FUNCTION_BLOCK CylinderVSensValve (* Composite Function Block Type *)
  (* Standard: 61499-2 *)
  (* Version 0.0, 5/29/2016, Andrei, nxtControl GmbH, template *)
  PACKAGE Main;
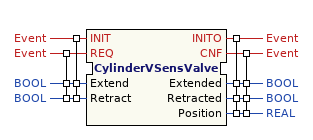
  EVENT_INPUT
    INIT WITH Extend, Retract; (* Initialization Request *)
    REQ WITH Extend, Retract; (* Normal Execution Request *)
  END_EVENT
  EVENT_OUTPUT
    INITO WITH Extended, Retracted, Position; (* Initialization Confirm *)
    CNF WITH Extended, Retracted, Position; (* Execution Confirmation *)
  END_EVENT
  VAR_INPUT
    Extend : BOOL; (* Input event qualifier *)
    Retract : BOOL;
  END_VAR
  VAR_OUTPUT
    Extended : BOOL; (* Output event qualifier *)
    Retracted : BOOL;
    Position : REAL;
  END_VAR
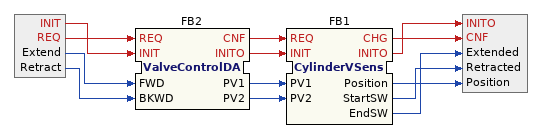
  FBS
    FB2 : ValveControlDA;
    FB1 : CylinderVSens;
  END_FBS
  EVENT_CONNECTIONS
    REQ TO FB2.REQ;
    INIT TO FB2.INIT;
    FB2.CNF TO FB1.REQ;
    FB1.CHG TO CNF;
    FB1.INITO TO INITO;
    FB2.INITO TO FB1.INIT;
  END_CONNECTIONS
  DATA_CONNECTIONS
    Extend TO FB2.FWD;
    Retract TO FB2.BKWD;
    FB2.PV1 TO FB1.PV1;
    FB2.PV2 TO FB1.PV2;
    FB1.Position TO Position;
    FB1.StartSW TO Retracted;
    FB1.EndSW TO Extended;
  END_CONNECTIONS
END_FUNCTION_BLOCK
